REGION Network 57: Step[420] : GapPad Down
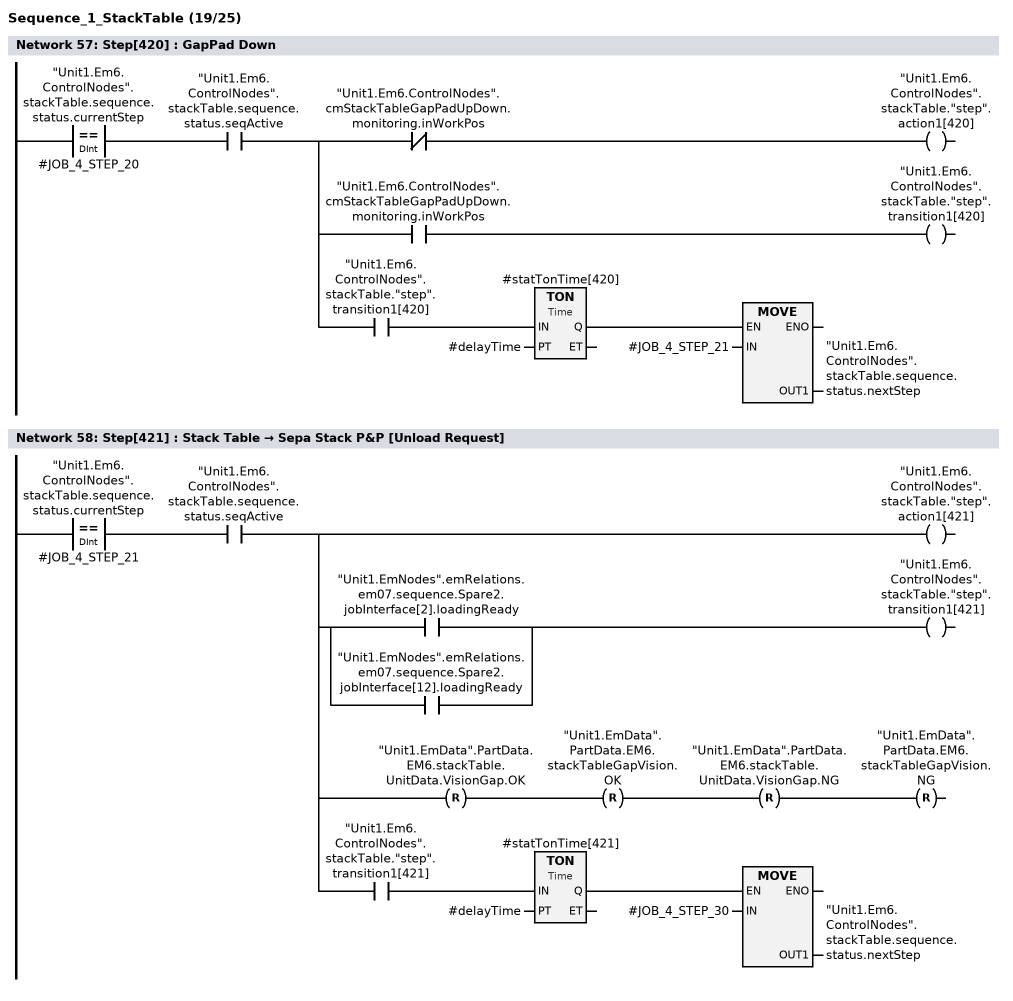
   RUNG wire#powerrail
      { S7_Templates := "SrcType := DInt" } EQ_Contact(in1 := "Unit1.Em6.ControlNodes".stackTable.sequence.status.currentStep, in2 := #JOB_4_STEP_20)
      Contact( "Unit1.Em6.ControlNodes".stackTable.sequence.status.seqActive )
      wire#w1
      I_Contact( "Unit1.Em6.ControlNodes".cmStackTableGapPadUpDown.monitoring.inWorkPos )
      Coil( "Unit1.Em6.ControlNodes".stackTable."step".action1[420] )
   END_RUNG
   RUNG wire#w1
      Contact( "Unit1.Em6.ControlNodes".cmStackTableGapPadUpDown.monitoring.inWorkPos )
      Coil( "Unit1.Em6.ControlNodes".stackTable."step".transition1[420] )
   END_RUNG
   RUNG wire#w1
      Contact( "Unit1.Em6.ControlNodes".stackTable."step".transition1[420] )
      { S7_Templates := "time_type := Time" } #statTonTime[420].TON(pt := #delayTime, et =>)
      Move(in := #JOB_4_STEP_21, out1 => "Unit1.Em6.ControlNodes".stackTable.sequence.status.nextStep)
   END_RUNG
   // the same network as SCL:
   #_w1 := ("Unit1.Em6.ControlNodes".stackTable.sequence.status.currentStep = #JOB_4_STEP_20) AND "Unit1.Em6.ControlNodes".stackTable.sequence.status.seqActive;
   "Unit1.Em6.ControlNodes".stackTable."step".action1[420] := #_w1 AND NOT "Unit1.Em6.ControlNodes".cmStackTableGapPadUpDown.monitoring.inWorkPos;
   "Unit1.Em6.ControlNodes".stackTable."step".transition1[420] := #_w1 AND "Unit1.Em6.ControlNodes".cmStackTableGapPadUpDown.monitoring.inWorkPos;
   #statTonTime[420].TON(IN := #_w1 AND "Unit1.Em6.ControlNodes".stackTable."step".transition1[420],
                         PT := #delayTime);
   IF #statTonTime[420].Q THEN
       "Unit1.Em6.ControlNodes".stackTable.sequence.status.nextStep := #JOB_4_STEP_21;
   END_IF;
END_REGION

REGION Network 58: Step[421] : Stack Table → Sepa Stack P&P [Unload Request]
   RUNG wire#powerrail
      { S7_Templates := "SrcType := DInt" } EQ_Contact(in1 := "Unit1.Em6.ControlNodes".stackTable.sequence.status.currentStep, in2 := #JOB_4_STEP_21)
      Contact( "Unit1.Em6.ControlNodes".stackTable.sequence.status.seqActive )
      wire#w1
      Coil( "Unit1.Em6.ControlNodes".stackTable."step".action1[421] )
   END_RUNG
   RUNG wire#w1
      Contact( "Unit1.EmNodes".emRelations.em07.sequence.Spare2.jobInterface[2].loadingReady )
      wire#w2
      Coil( "Unit1.Em6.ControlNodes".stackTable."step".transition1[421] )
   END_RUNG
   RUNG wire#w1
      Contact( "Unit1.EmNodes".emRelations.em07.sequence.Spare2.jobInterface[12].loadingReady )
   END_RUNG wire#w2
   RUNG wire#w1
      R_Coil( "Unit1.EmData".PartData.EM6.stackTable.UnitData.VisionGap.OK )
      R_Coil( "Unit1.EmData".PartData.EM6.stackTableGapVision.OK )
      R_Coil( "Unit1.EmData".PartData.EM6.stackTable.UnitData.VisionGap.NG )
      R_Coil( "Unit1.EmData".PartData.EM6.stackTableGapVision.NG )
   END_RUNG
   RUNG wire#w1
      Contact( "Unit1.Em6.ControlNodes".stackTable."step".transition1[421] )
      { S7_Templates := "time_type := Time" } #statTonTime[421].TON(pt := #delayTime, et =>)
      Move(in := #JOB_4_STEP_30, out1 => "Unit1.Em6.ControlNodes".stackTable.sequence.status.nextStep)
   END_RUNG
   // the same network as SCL:
   "Unit1.Em6.ControlNodes".stackTable."step".action1[421] := ("Unit1.Em6.ControlNodes".stackTable.sequence.status.currentStep = #JOB_4_STEP_21) AND "Unit1.Em6.ControlNodes".stackTable.sequence.status.seqActive;
   "Unit1.Em6.ControlNodes".stackTable."step".transition1[421] := ("Unit1.Em6.ControlNodes".stackTable.sequence.status.currentStep = #JOB_4_STEP_21) AND "Unit1.Em6.ControlNodes".stackTable.sequence.status.seqActive AND ("Unit1.EmNodes".emRelations.em07.sequence.Spare2.jobInterface[2].loadingReady OR "Unit1.EmNodes".emRelations.em07.sequence.Spare2.jobInterface[12].loadingReady);
   IF ("Unit1.Em6.ControlNodes".stackTable.sequence.status.currentStep = #JOB_4_STEP_21) AND "Unit1.Em6.ControlNodes".stackTable.sequence.status.seqActive THEN
       "Unit1.EmData".PartData.EM6.stackTable.UnitData.VisionGap.OK := FALSE;
       "Unit1.EmData".PartData.EM6.stackTableGapVision.OK := FALSE;
       "Unit1.EmData".PartData.EM6.stackTable.UnitData.VisionGap.NG := FALSE;
       "Unit1.EmData".PartData.EM6.stackTableGapVision.NG := FALSE;
   END_IF;
   #statTonTime[421].TON(IN := ("Unit1.Em6.ControlNodes".stackTable.sequence.status.currentStep = #JOB_4_STEP_21) AND "Unit1.Em6.ControlNodes".stackTable.sequence.status.seqActive AND "Unit1.Em6.ControlNodes".stackTable."step".transition1[421],
                         PT := #delayTime);
   IF #statTonTime[421].Q THEN
       "Unit1.Em6.ControlNodes".stackTable.sequence.status.nextStep := #JOB_4_STEP_30;
   END_IF;
END_REGION

REGION Network 59: Step[430] : A,C.Mendrel Y,Z-Axis Wait Pos
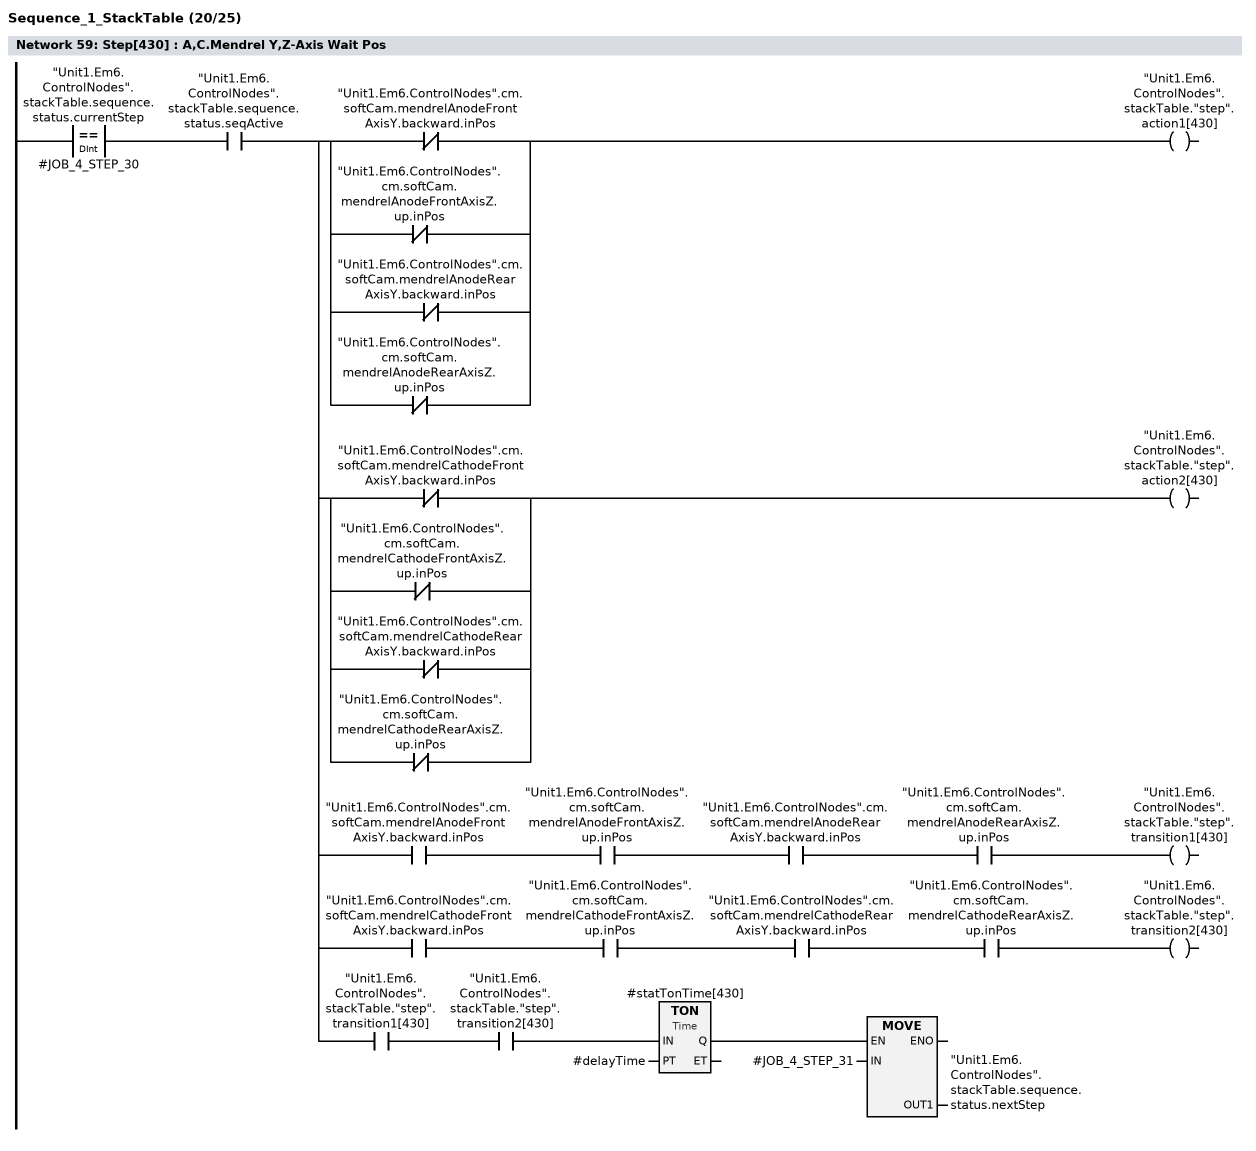
   RUNG wire#powerrail
      { S7_Templates := "SrcType := DInt" } EQ_Contact(in1 := "Unit1.Em6.ControlNodes".stackTable.sequence.status.currentStep, in2 := #JOB_4_STEP_30)
      Contact( "Unit1.Em6.ControlNodes".stackTable.sequence.status.seqActive )
      wire#w1
      I_Contact( "Unit1.Em6.ControlNodes".cm.softCam.mendrelAnodeFrontAxisY.backward.inPos )
      wire#w2
      Coil( "Unit1.Em6.ControlNodes".stackTable."step".action1[430] )
   END_RUNG
   RUNG wire#w1
      I_Contact( "Unit1.Em6.ControlNodes".cm.softCam.mendrelAnodeFrontAxisZ.up.inPos )
   END_RUNG wire#w2
   RUNG wire#w1
      I_Contact( "Unit1.Em6.ControlNodes".cm.softCam.mendrelAnodeRearAxisY.backward.inPos )
   END_RUNG wire#w2
   RUNG wire#w1
      I_Contact( "Unit1.Em6.ControlNodes".cm.softCam.mendrelAnodeRearAxisZ.up.inPos )
   END_RUNG wire#w2
   RUNG wire#w1
      I_Contact( "Unit1.Em6.ControlNodes".cm.softCam.mendrelCathodeFrontAxisY.backward.inPos )
      wire#w3
      Coil( "Unit1.Em6.ControlNodes".stackTable."step".action2[430] )
   END_RUNG
   RUNG wire#w1
      I_Contact( "Unit1.Em6.ControlNodes".cm.softCam.mendrelCathodeFrontAxisZ.up.inPos )
   END_RUNG wire#w3
   RUNG wire#w1
      I_Contact( "Unit1.Em6.ControlNodes".cm.softCam.mendrelCathodeRearAxisY.backward.inPos )
   END_RUNG wire#w3
   RUNG wire#w1
      I_Contact( "Unit1.Em6.ControlNodes".cm.softCam.mendrelCathodeRearAxisZ.up.inPos )
   END_RUNG wire#w3
   RUNG wire#w1
      Contact( "Unit1.Em6.ControlNodes".cm.softCam.mendrelAnodeFrontAxisY.backward.inPos )
      Contact( "Unit1.Em6.ControlNodes".cm.softCam.mendrelAnodeFrontAxisZ.up.inPos )
      Contact( "Unit1.Em6.ControlNodes".cm.softCam.mendrelAnodeRearAxisY.backward.inPos )
      Contact( "Unit1.Em6.ControlNodes".cm.softCam.mendrelAnodeRearAxisZ.up.inPos )
      Coil( "Unit1.Em6.ControlNodes".stackTable."step".transition1[430] )
   END_RUNG
   RUNG wire#w1
      Contact( "Unit1.Em6.ControlNodes".cm.softCam.mendrelCathodeFrontAxisY.backward.inPos )
      Contact( "Unit1.Em6.ControlNodes".cm.softCam.mendrelCathodeFrontAxisZ.up.inPos )
      Contact( "Unit1.Em6.ControlNodes".cm.softCam.mendrelCathodeRearAxisY.backward.inPos )
      Contact( "Unit1.Em6.ControlNodes".cm.softCam.mendrelCathodeRearAxisZ.up.inPos )
      Coil( "Unit1.Em6.ControlNodes".stackTable."step".transition2[430] )
   END_RUNG
   RUNG wire#w1
      Contact( "Unit1.Em6.ControlNodes".stackTable."step".transition1[430] )
      Contact( "Unit1.Em6.ControlNodes".stackTable."step".transition2[430] )
      { S7_Templates := "time_type := Time" } #statTonTime[430].TON(pt := #delayTime, et =>)
      Move(in := #JOB_4_STEP_31, out1 => "Unit1.Em6.ControlNodes".stackTable.sequence.status.nextStep)
   END_RUNG
   // the same network as SCL:
   #_w1 := ("Unit1.Em6.ControlNodes".stackTable.sequence.status.currentStep = #JOB_4_STEP_30) AND "Unit1.Em6.ControlNodes".stackTable.sequence.status.seqActive;
   "Unit1.Em6.ControlNodes".stackTable."step".action1[430] := #_w1 AND (NOT "Unit1.Em6.ControlNodes".cm.softCam.mendrelAnodeFrontAxisY.backward.inPos OR NOT "Unit1.Em6.ControlNodes".cm.softCam.mendrelAnodeFrontAxisZ.up.inPos OR NOT "Unit1.Em6.ControlNodes".cm.softCam.mendrelAnodeRearAxisY.backward.inPos OR NOT "Unit1.Em6.ControlNodes".cm.softCam.mendrelAnodeRearAxisZ.up.inPos);
   "Unit1.Em6.ControlNodes".stackTable."step".action2[430] := #_w1 AND (NOT "Unit1.Em6.ControlNodes".cm.softCam.mendrelCathodeFrontAxisY.backward.inPos OR NOT "Unit1.Em6.ControlNodes".cm.softCam.mendrelCathodeFrontAxisZ.up.inPos OR NOT "Unit1.Em6.ControlNodes".cm.softCam.mendrelCathodeRearAxisY.backward.inPos OR NOT "Unit1.Em6.ControlNodes".cm.softCam.mendrelCathodeRearAxisZ.up.inPos);
   "Unit1.Em6.ControlNodes".stackTable."step".transition1[430] := #_w1 AND "Unit1.Em6.ControlNodes".cm.softCam.mendrelAnodeFrontAxisY.backward.inPos AND "Unit1.Em6.ControlNodes".cm.softCam.mendrelAnodeFrontAxisZ.up.inPos AND "Unit1.Em6.ControlNodes".cm.softCam.mendrelAnodeRearAxisY.backward.inPos AND "Unit1.Em6.ControlNodes".cm.softCam.mendrelAnodeRearAxisZ.up.inPos;
   "Unit1.Em6.ControlNodes".stackTable."step".transition2[430] := #_w1 AND "Unit1.Em6.ControlNodes".cm.softCam.mendrelCathodeFrontAxisY.backward.inPos AND "Unit1.Em6.ControlNodes".cm.softCam.mendrelCathodeFrontAxisZ.up.inPos AND "Unit1.Em6.ControlNodes".cm.softCam.mendrelCathodeRearAxisY.backward.inPos AND "Unit1.Em6.ControlNodes".cm.softCam.mendrelCathodeRearAxisZ.up.inPos;
   #statTonTime[430].TON(IN := #_w1 AND "Unit1.Em6.ControlNodes".stackTable."step".transition1[430] AND "Unit1.Em6.ControlNodes".stackTable."step".transition2[430],
                         PT := #delayTime);
   IF #statTonTime[430].Q THEN
       "Unit1.Em6.ControlNodes".stackTable.sequence.status.nextStep := #JOB_4_STEP_31;
   END_IF;
END_REGION

REGION Network 60: Step[431] : Stack Table → Sepa Stack P&P [Unclamp Done]
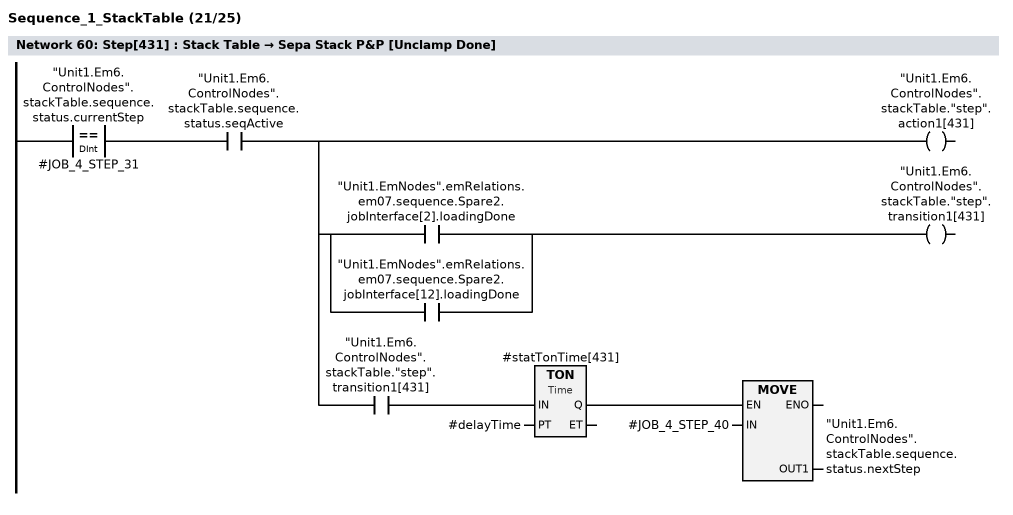
   RUNG wire#powerrail
      { S7_Templates := "SrcType := DInt" } EQ_Contact(in1 := "Unit1.Em6.ControlNodes".stackTable.sequence.status.currentStep, in2 := #JOB_4_STEP_31)
      Contact( "Unit1.Em6.ControlNodes".stackTable.sequence.status.seqActive )
      wire#w1
      Coil( "Unit1.Em6.ControlNodes".stackTable."step".action1[431] )
   END_RUNG
   RUNG wire#w1
      Contact( "Unit1.EmNodes".emRelations.em07.sequence.Spare2.jobInterface[2].loadingDone )
      wire#w2
      Coil( "Unit1.Em6.ControlNodes".stackTable."step".transition1[431] )
   END_RUNG
   RUNG wire#w1
      Contact( "Unit1.EmNodes".emRelations.em07.sequence.Spare2.jobInterface[12].loadingDone )
   END_RUNG wire#w2
   RUNG wire#w1
      Contact( "Unit1.Em6.ControlNodes".stackTable."step".transition1[431] )
      { S7_Templates := "time_type := Time" } #statTonTime[431].TON(pt := #delayTime, et =>)
      Move(in := #JOB_4_STEP_40, out1 => "Unit1.Em6.ControlNodes".stackTable.sequence.status.nextStep)
   END_RUNG
   // the same network as SCL:
   "Unit1.Em6.ControlNodes".stackTable."step".action1[431] := ("Unit1.Em6.ControlNodes".stackTable.sequence.status.currentStep = #JOB_4_STEP_31) AND "Unit1.Em6.ControlNodes".stackTable.sequence.status.seqActive;
   "Unit1.Em6.ControlNodes".stackTable."step".transition1[431] := ("Unit1.Em6.ControlNodes".stackTable.sequence.status.currentStep = #JOB_4_STEP_31) AND "Unit1.Em6.ControlNodes".stackTable.sequence.status.seqActive AND ("Unit1.EmNodes".emRelations.em07.sequence.Spare2.jobInterface[2].loadingDone OR "Unit1.EmNodes".emRelations.em07.sequence.Spare2.jobInterface[12].loadingDone);
   #statTonTime[431].TON(IN := ("Unit1.Em6.ControlNodes".stackTable.sequence.status.currentStep = #JOB_4_STEP_31) AND "Unit1.Em6.ControlNodes".stackTable.sequence.status.seqActive AND "Unit1.Em6.ControlNodes".stackTable."step".transition1[431],
                         PT := #delayTime);
   IF #statTonTime[431].Q THEN
       "Unit1.Em6.ControlNodes".stackTable.sequence.status.nextStep := #JOB_4_STEP_40;
   END_IF;
END_REGION

REGION Network 61: Step[440] : A,C.Mendrel Y,Z-Axis Work Pos
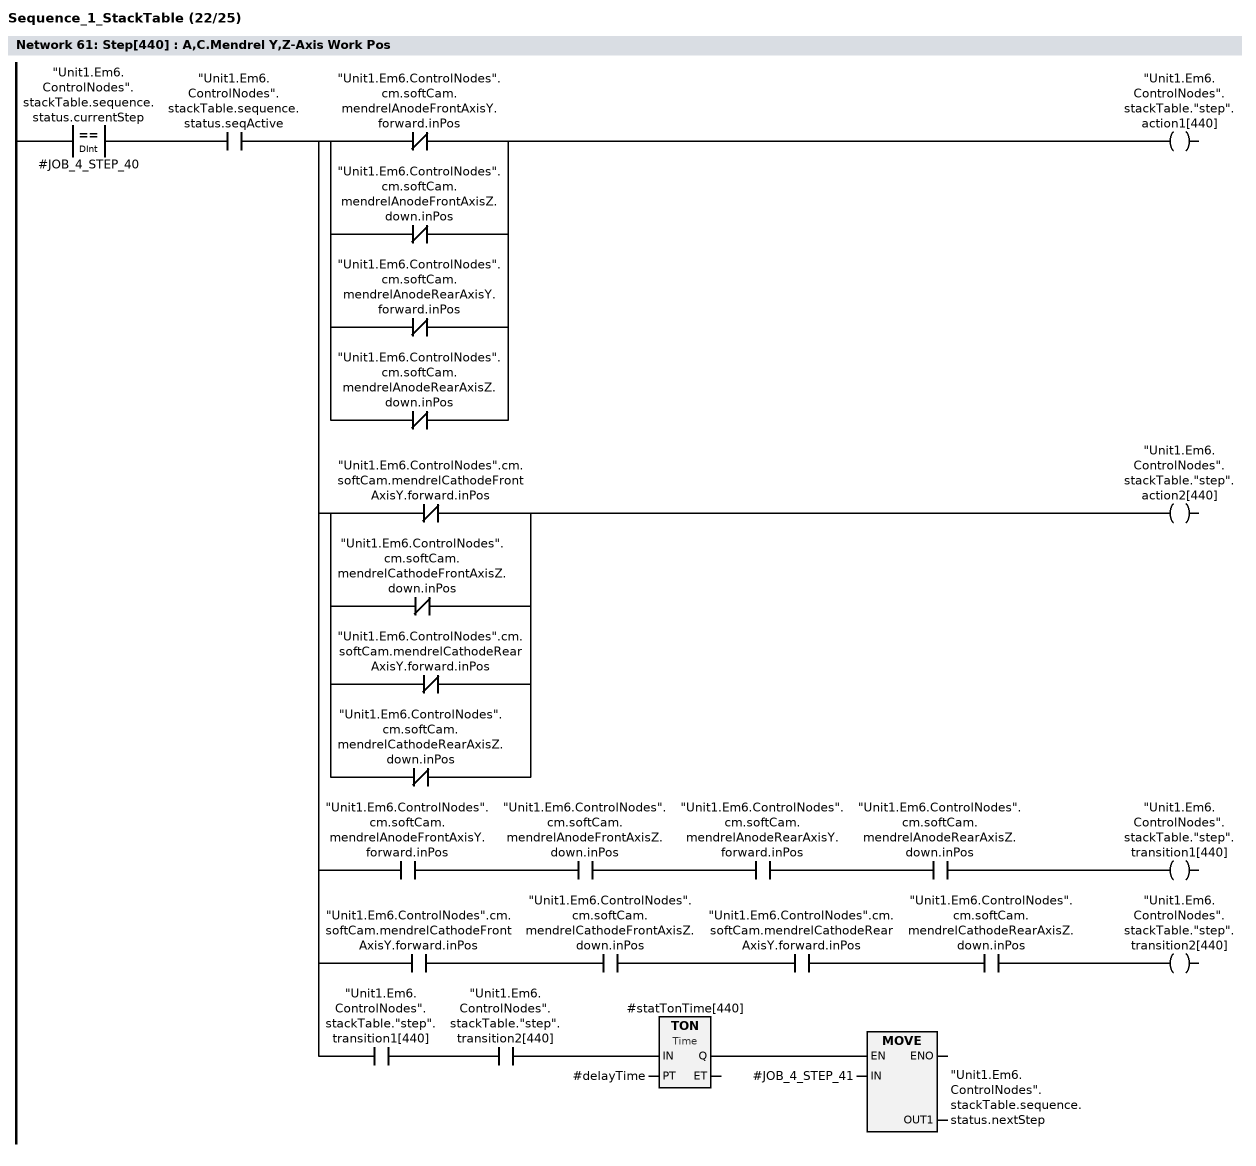
   RUNG wire#powerrail
      { S7_Templates := "SrcType := DInt" } EQ_Contact(in1 := "Unit1.Em6.ControlNodes".stackTable.sequence.status.currentStep, in2 := #JOB_4_STEP_40)
      Contact( "Unit1.Em6.ControlNodes".stackTable.sequence.status.seqActive )
      wire#w1
      I_Contact( "Unit1.Em6.ControlNodes".cm.softCam.mendrelAnodeFrontAxisY.forward.inPos )
      wire#w2
      Coil( "Unit1.Em6.ControlNodes".stackTable."step".action1[440] )
   END_RUNG
   RUNG wire#w1
      I_Contact( "Unit1.Em6.ControlNodes".cm.softCam.mendrelAnodeFrontAxisZ.down.inPos )
   END_RUNG wire#w2
   RUNG wire#w1
      I_Contact( "Unit1.Em6.ControlNodes".cm.softCam.mendrelAnodeRearAxisY.forward.inPos )
   END_RUNG wire#w2
   RUNG wire#w1
      I_Contact( "Unit1.Em6.ControlNodes".cm.softCam.mendrelAnodeRearAxisZ.down.inPos )
   END_RUNG wire#w2
   RUNG wire#w1
      I_Contact( "Unit1.Em6.ControlNodes".cm.softCam.mendrelCathodeFrontAxisY.forward.inPos )
      wire#w3
      Coil( "Unit1.Em6.ControlNodes".stackTable."step".action2[440] )
   END_RUNG
   RUNG wire#w1
      I_Contact( "Unit1.Em6.ControlNodes".cm.softCam.mendrelCathodeFrontAxisZ.down.inPos )
   END_RUNG wire#w3
   RUNG wire#w1
      I_Contact( "Unit1.Em6.ControlNodes".cm.softCam.mendrelCathodeRearAxisY.forward.inPos )
   END_RUNG wire#w3
   RUNG wire#w1
      I_Contact( "Unit1.Em6.ControlNodes".cm.softCam.mendrelCathodeRearAxisZ.down.inPos )
   END_RUNG wire#w3
   RUNG wire#w1
      Contact( "Unit1.Em6.ControlNodes".cm.softCam.mendrelAnodeFrontAxisY.forward.inPos )
      Contact( "Unit1.Em6.ControlNodes".cm.softCam.mendrelAnodeFrontAxisZ.down.inPos )
      Contact( "Unit1.Em6.ControlNodes".cm.softCam.mendrelAnodeRearAxisY.forward.inPos )
      Contact( "Unit1.Em6.ControlNodes".cm.softCam.mendrelAnodeRearAxisZ.down.inPos )
      Coil( "Unit1.Em6.ControlNodes".stackTable."step".transition1[440] )
   END_RUNG
   RUNG wire#w1
      Contact( "Unit1.Em6.ControlNodes".cm.softCam.mendrelCathodeFrontAxisY.forward.inPos )
      Contact( "Unit1.Em6.ControlNodes".cm.softCam.mendrelCathodeFrontAxisZ.down.inPos )
      Contact( "Unit1.Em6.ControlNodes".cm.softCam.mendrelCathodeRearAxisY.forward.inPos )
      Contact( "Unit1.Em6.ControlNodes".cm.softCam.mendrelCathodeRearAxisZ.down.inPos )
      Coil( "Unit1.Em6.ControlNodes".stackTable."step".transition2[440] )
   END_RUNG
   RUNG wire#w1
      Contact( "Unit1.Em6.ControlNodes".stackTable."step".transition1[440] )
      Contact( "Unit1.Em6.ControlNodes".stackTable."step".transition2[440] )
      { S7_Templates := "time_type := Time" } #statTonTime[440].TON(pt := #delayTime, et =>)
      Move(in := #JOB_4_STEP_41, out1 => "Unit1.Em6.ControlNodes".stackTable.sequence.status.nextStep)
   END_RUNG
   // the same network as SCL:
   #_w1 := ("Unit1.Em6.ControlNodes".stackTable.sequence.status.currentStep = #JOB_4_STEP_40) AND "Unit1.Em6.ControlNodes".stackTable.sequence.status.seqActive;
   "Unit1.Em6.ControlNodes".stackTable."step".action1[440] := #_w1 AND (NOT "Unit1.Em6.ControlNodes".cm.softCam.mendrelAnodeFrontAxisY.forward.inPos OR NOT "Unit1.Em6.ControlNodes".cm.softCam.mendrelAnodeFrontAxisZ.down.inPos OR NOT "Unit1.Em6.ControlNodes".cm.softCam.mendrelAnodeRearAxisY.forward.inPos OR NOT "Unit1.Em6.ControlNodes".cm.softCam.mendrelAnodeRearAxisZ.down.inPos);
   "Unit1.Em6.ControlNodes".stackTable."step".action2[440] := #_w1 AND (NOT "Unit1.Em6.ControlNodes".cm.softCam.mendrelCathodeFrontAxisY.forward.inPos OR NOT "Unit1.Em6.ControlNodes".cm.softCam.mendrelCathodeFrontAxisZ.down.inPos OR NOT "Unit1.Em6.ControlNodes".cm.softCam.mendrelCathodeRearAxisY.forward.inPos OR NOT "Unit1.Em6.ControlNodes".cm.softCam.mendrelCathodeRearAxisZ.down.inPos);
   "Unit1.Em6.ControlNodes".stackTable."step".transition1[440] := #_w1 AND "Unit1.Em6.ControlNodes".cm.softCam.mendrelAnodeFrontAxisY.forward.inPos AND "Unit1.Em6.ControlNodes".cm.softCam.mendrelAnodeFrontAxisZ.down.inPos AND "Unit1.Em6.ControlNodes".cm.softCam.mendrelAnodeRearAxisY.forward.inPos AND "Unit1.Em6.ControlNodes".cm.softCam.mendrelAnodeRearAxisZ.down.inPos;
   "Unit1.Em6.ControlNodes".stackTable."step".transition2[440] := #_w1 AND "Unit1.Em6.ControlNodes".cm.softCam.mendrelCathodeFrontAxisY.forward.inPos AND "Unit1.Em6.ControlNodes".cm.softCam.mendrelCathodeFrontAxisZ.down.inPos AND "Unit1.Em6.ControlNodes".cm.softCam.mendrelCathodeRearAxisY.forward.inPos AND "Unit1.Em6.ControlNodes".cm.softCam.mendrelCathodeRearAxisZ.down.inPos;
   #statTonTime[440].TON(IN := #_w1 AND "Unit1.Em6.ControlNodes".stackTable."step".transition1[440] AND "Unit1.Em6.ControlNodes".stackTable."step".transition2[440],
                         PT := #delayTime);
   IF #statTonTime[440].Q THEN
       "Unit1.Em6.ControlNodes".stackTable.sequence.status.nextStep := #JOB_4_STEP_41;
   END_IF;
END_REGION

REGION Network 62: Step[441] : Stack Table → Sepa Stack P&P [Clamp Done]
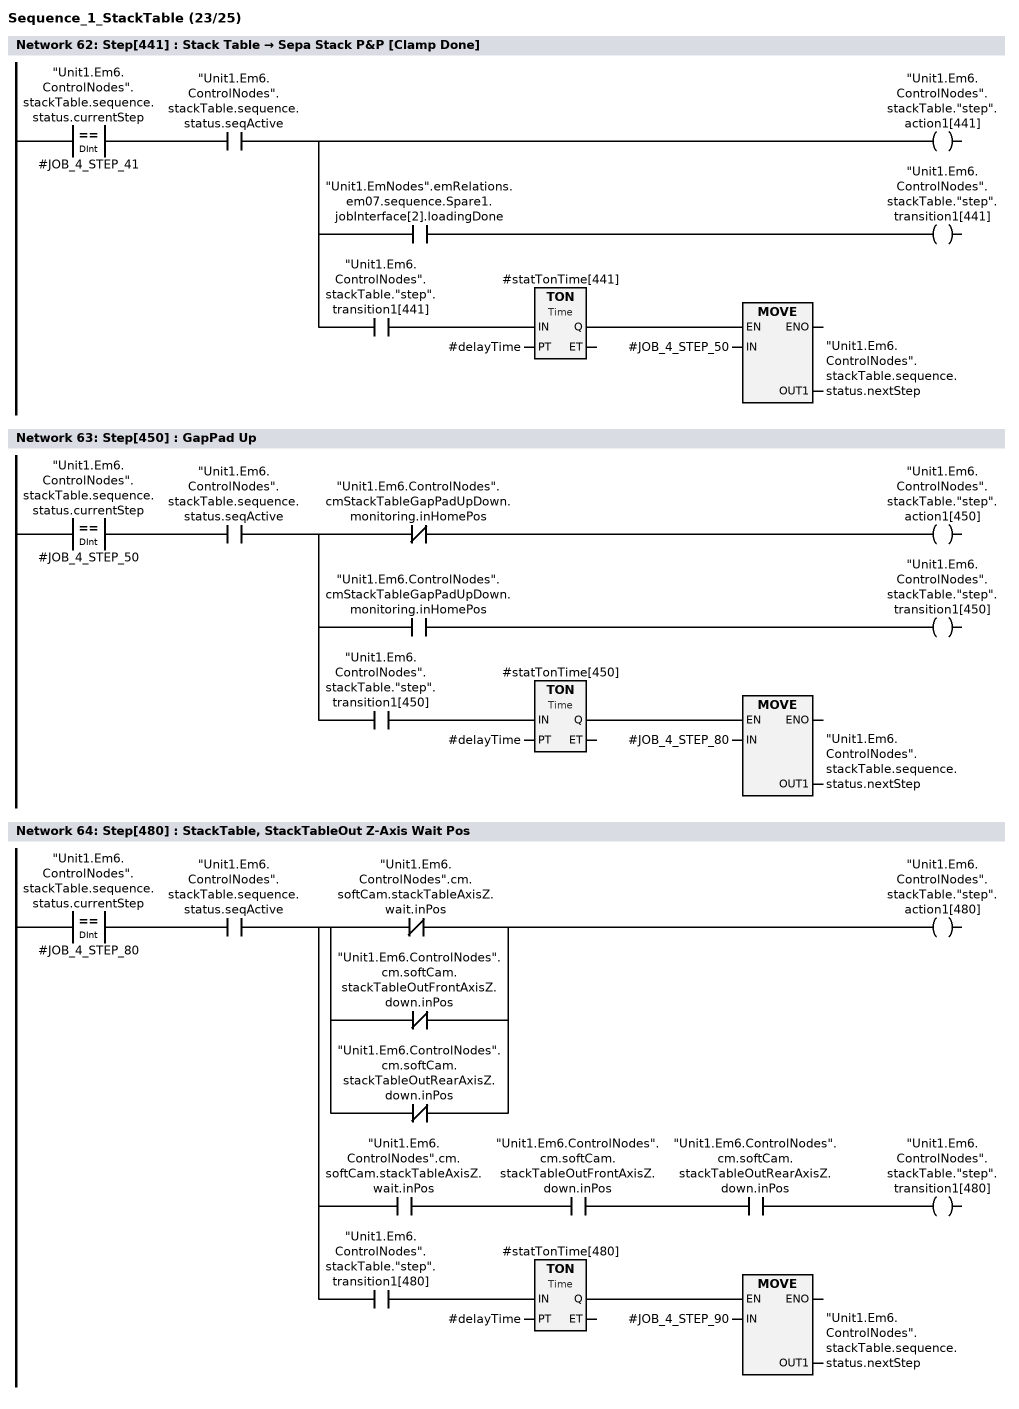
   RUNG wire#powerrail
      { S7_Templates := "SrcType := DInt" } EQ_Contact(in1 := "Unit1.Em6.ControlNodes".stackTable.sequence.status.currentStep, in2 := #JOB_4_STEP_41)
      Contact( "Unit1.Em6.ControlNodes".stackTable.sequence.status.seqActive )
      wire#w1
      Coil( "Unit1.Em6.ControlNodes".stackTable."step".action1[441] )
   END_RUNG
   RUNG wire#w1
      Contact( "Unit1.EmNodes".emRelations.em07.sequence.Spare1.jobInterface[2].loadingDone )
      Coil( "Unit1.Em6.ControlNodes".stackTable."step".transition1[441] )
   END_RUNG
   RUNG wire#w1
      Contact( "Unit1.Em6.ControlNodes".stackTable."step".transition1[441] )
      { S7_Templates := "time_type := Time" } #statTonTime[441].TON(pt := #delayTime, et =>)
      Move(in := #JOB_4_STEP_50, out1 => "Unit1.Em6.ControlNodes".stackTable.sequence.status.nextStep)
   END_RUNG
   // the same network as SCL:
   "Unit1.Em6.ControlNodes".stackTable."step".action1[441] := ("Unit1.Em6.ControlNodes".stackTable.sequence.status.currentStep = #JOB_4_STEP_41) AND "Unit1.Em6.ControlNodes".stackTable.sequence.status.seqActive;
   "Unit1.Em6.ControlNodes".stackTable."step".transition1[441] := ("Unit1.Em6.ControlNodes".stackTable.sequence.status.currentStep = #JOB_4_STEP_41) AND "Unit1.Em6.ControlNodes".stackTable.sequence.status.seqActive AND "Unit1.EmNodes".emRelations.em07.sequence.Spare1.jobInterface[2].loadingDone;
   #statTonTime[441].TON(IN := ("Unit1.Em6.ControlNodes".stackTable.sequence.status.currentStep = #JOB_4_STEP_41) AND "Unit1.Em6.ControlNodes".stackTable.sequence.status.seqActive AND "Unit1.Em6.ControlNodes".stackTable."step".transition1[441],
                         PT := #delayTime);
   IF #statTonTime[441].Q THEN
       "Unit1.Em6.ControlNodes".stackTable.sequence.status.nextStep := #JOB_4_STEP_50;
   END_IF;
END_REGION

REGION Network 63: Step[450] : GapPad Up
   RUNG wire#powerrail
      { S7_Templates := "SrcType := DInt" } EQ_Contact(in1 := "Unit1.Em6.ControlNodes".stackTable.sequence.status.currentStep, in2 := #JOB_4_STEP_50)
      Contact( "Unit1.Em6.ControlNodes".stackTable.sequence.status.seqActive )
      wire#w1
      I_Contact( "Unit1.Em6.ControlNodes".cmStackTableGapPadUpDown.monitoring.inHomePos )
      Coil( "Unit1.Em6.ControlNodes".stackTable."step".action1[450] )
   END_RUNG
   RUNG wire#w1
      Contact( "Unit1.Em6.ControlNodes".cmStackTableGapPadUpDown.monitoring.inHomePos )
      Coil( "Unit1.Em6.ControlNodes".stackTable."step".transition1[450] )
   END_RUNG
   RUNG wire#w1
      Contact( "Unit1.Em6.ControlNodes".stackTable."step".transition1[450] )
      { S7_Templates := "time_type := Time" } #statTonTime[450].TON(pt := #delayTime, et =>)
      Move(in := #JOB_4_STEP_80, out1 => "Unit1.Em6.ControlNodes".stackTable.sequence.status.nextStep)
   END_RUNG
   // the same network as SCL:
   #_w1 := ("Unit1.Em6.ControlNodes".stackTable.sequence.status.currentStep = #JOB_4_STEP_50) AND "Unit1.Em6.ControlNodes".stackTable.sequence.status.seqActive;
   "Unit1.Em6.ControlNodes".stackTable."step".action1[450] := #_w1 AND NOT "Unit1.Em6.ControlNodes".cmStackTableGapPadUpDown.monitoring.inHomePos;
   "Unit1.Em6.ControlNodes".stackTable."step".transition1[450] := #_w1 AND "Unit1.Em6.ControlNodes".cmStackTableGapPadUpDown.monitoring.inHomePos;
   #statTonTime[450].TON(IN := #_w1 AND "Unit1.Em6.ControlNodes".stackTable."step".transition1[450],
                         PT := #delayTime);
   IF #statTonTime[450].Q THEN
       "Unit1.Em6.ControlNodes".stackTable.sequence.status.nextStep := #JOB_4_STEP_80;
   END_IF;
END_REGION

REGION Network 64: Step[480] : StackTable, StackTableOut Z-Axis Wait Pos
   RUNG wire#powerrail
      { S7_Templates := "SrcType := DInt" } EQ_Contact(in1 := "Unit1.Em6.ControlNodes".stackTable.sequence.status.currentStep, in2 := #JOB_4_STEP_80)
      Contact( "Unit1.Em6.ControlNodes".stackTable.sequence.status.seqActive )
      wire#w1
      I_Contact( "Unit1.Em6.ControlNodes".cm.softCam.stackTableAxisZ.wait.inPos )
      wire#w2
      Coil( "Unit1.Em6.ControlNodes".stackTable."step".action1[480] )
   END_RUNG
   RUNG wire#w1
      I_Contact( "Unit1.Em6.ControlNodes".cm.softCam.stackTableOutFrontAxisZ.down.inPos )
   END_RUNG wire#w2
   RUNG wire#w1
      I_Contact( "Unit1.Em6.ControlNodes".cm.softCam.stackTableOutRearAxisZ.down.inPos )
   END_RUNG wire#w2
   RUNG wire#w1
      Contact( "Unit1.Em6.ControlNodes".cm.softCam.stackTableAxisZ.wait.inPos )
      Contact( "Unit1.Em6.ControlNodes".cm.softCam.stackTableOutFrontAxisZ.down.inPos )
      Contact( "Unit1.Em6.ControlNodes".cm.softCam.stackTableOutRearAxisZ.down.inPos )
      Coil( "Unit1.Em6.ControlNodes".stackTable."step".transition1[480] )
   END_RUNG
   RUNG wire#w1
      Contact( "Unit1.Em6.ControlNodes".stackTable."step".transition1[480] )
      { S7_Templates := "time_type := Time" } #statTonTime[480].TON(pt := #delayTime, et =>)
      Move(in := #JOB_4_STEP_90, out1 => "Unit1.Em6.ControlNodes".stackTable.sequence.status.nextStep)
   END_RUNG
   // the same network as SCL:
   #_w1 := ("Unit1.Em6.ControlNodes".stackTable.sequence.status.currentStep = #JOB_4_STEP_80) AND "Unit1.Em6.ControlNodes".stackTable.sequence.status.seqActive;
   "Unit1.Em6.ControlNodes".stackTable."step".action1[480] := #_w1 AND (NOT "Unit1.Em6.ControlNodes".cm.softCam.stackTableAxisZ.wait.inPos OR NOT "Unit1.Em6.ControlNodes".cm.softCam.stackTableOutFrontAxisZ.down.inPos OR NOT "Unit1.Em6.ControlNodes".cm.softCam.stackTableOutRearAxisZ.down.inPos);
   "Unit1.Em6.ControlNodes".stackTable."step".transition1[480] := #_w1 AND "Unit1.Em6.ControlNodes".cm.softCam.stackTableAxisZ.wait.inPos AND "Unit1.Em6.ControlNodes".cm.softCam.stackTableOutFrontAxisZ.down.inPos AND "Unit1.Em6.ControlNodes".cm.softCam.stackTableOutRearAxisZ.down.inPos;
   #statTonTime[480].TON(IN := #_w1 AND "Unit1.Em6.ControlNodes".stackTable."step".transition1[480],
                         PT := #delayTime);
   IF #statTonTime[480].Q THEN
       "Unit1.Em6.ControlNodes".stackTable.sequence.status.nextStep := #JOB_4_STEP_90;
   END_IF;
END_REGION

REGION Network 65: Step[490] : JOB[4] Step End
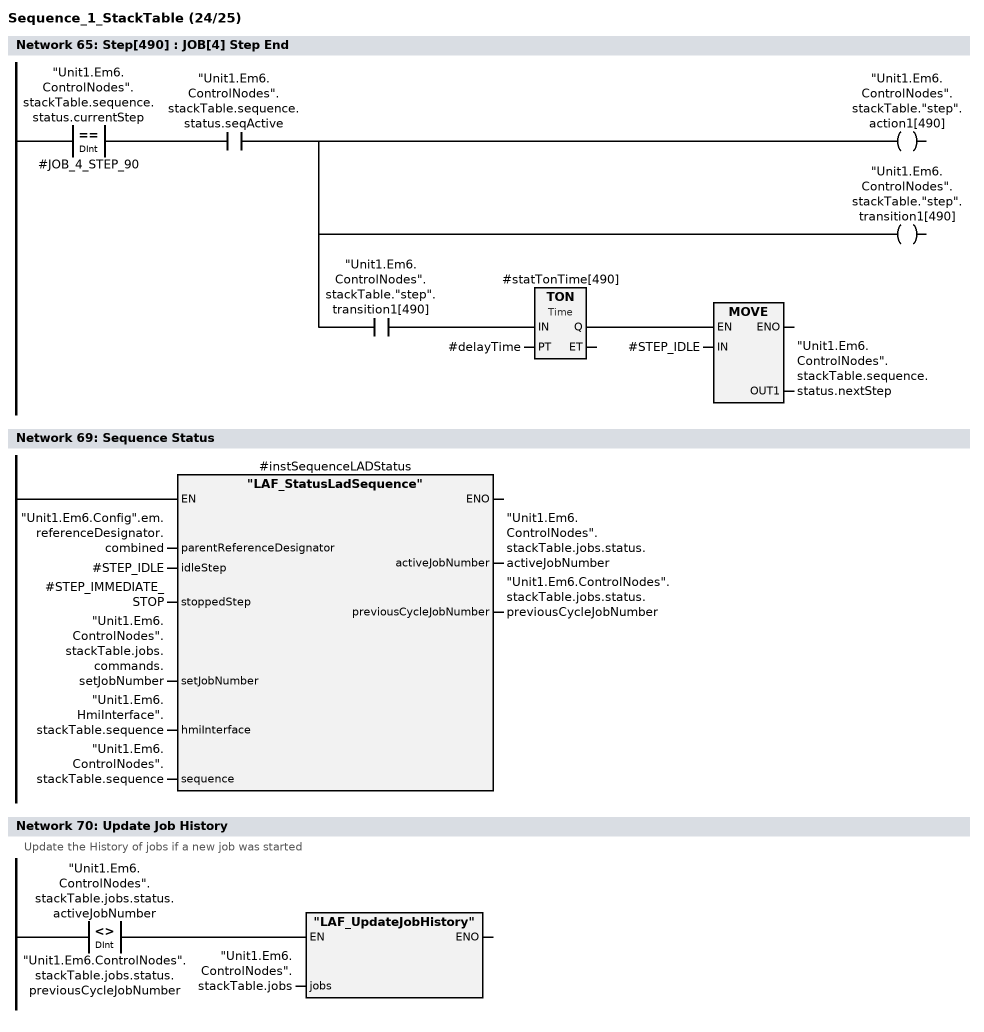
   RUNG wire#powerrail
      { S7_Templates := "SrcType := DInt" } EQ_Contact(in1 := "Unit1.Em6.ControlNodes".stackTable.sequence.status.currentStep, in2 := #JOB_4_STEP_90)
      Contact( "Unit1.Em6.ControlNodes".stackTable.sequence.status.seqActive )
      wire#w1
      Coil( "Unit1.Em6.ControlNodes".stackTable."step".action1[490] )
   END_RUNG
   RUNG wire#w1
      Coil( "Unit1.Em6.ControlNodes".stackTable."step".transition1[490] )
   END_RUNG
   RUNG wire#w1
      Contact( "Unit1.Em6.ControlNodes".stackTable."step".transition1[490] )
      { S7_Templates := "time_type := Time" } #statTonTime[490].TON(pt := #delayTime, et =>)
      Move(in := #STEP_IDLE, out1 => "Unit1.Em6.ControlNodes".stackTable.sequence.status.nextStep)
   END_RUNG
   // the same network as SCL:
   "Unit1.Em6.ControlNodes".stackTable."step".action1[490] := ("Unit1.Em6.ControlNodes".stackTable.sequence.status.currentStep = #JOB_4_STEP_90) AND "Unit1.Em6.ControlNodes".stackTable.sequence.status.seqActive;
   "Unit1.Em6.ControlNodes".stackTable."step".transition1[490] := ("Unit1.Em6.ControlNodes".stackTable.sequence.status.currentStep = #JOB_4_STEP_90) AND "Unit1.Em6.ControlNodes".stackTable.sequence.status.seqActive;
   #statTonTime[490].TON(IN := ("Unit1.Em6.ControlNodes".stackTable.sequence.status.currentStep = #JOB_4_STEP_90) AND "Unit1.Em6.ControlNodes".stackTable.sequence.status.seqActive AND "Unit1.Em6.ControlNodes".stackTable."step".transition1[490],
                         PT := #delayTime);
   IF #statTonTime[490].Q THEN
       "Unit1.Em6.ControlNodes".stackTable.sequence.status.nextStep := #STEP_IDLE;
   END_IF;
END_REGION

REGION Network 66: *************** IMMEDIATE STOP **************************
END_REGION

REGION Network 67: Immediate Stop
END_REGION

REGION Network 68: *************** Status updates **************************
END_REGION

REGION Network 69: Sequence Status
   RUNG wire#powerrail
      #instSequenceLADStatus(parentReferenceDesignator := "Unit1.Em6.Config".em.referenceDesignator.combined, idleStep := #STEP_IDLE, stoppedStep := #STEP_IMMEDIATE_STOP, setJobNumber := "Unit1.Em6.ControlNodes".stackTable.jobs.commands.setJobNumber, hmiInterface := "Unit1.Em6.HmiInterface".stackTable.sequence, sequence := "Unit1.Em6.ControlNodes".stackTable.sequence, activeJobNumber => "Unit1.Em6.ControlNodes".stackTable.jobs.status.activeJobNumber, previousCycleJobNumber => "Unit1.Em6.ControlNodes".stackTable.jobs.status.previousCycleJobNumber)
   END_RUNG
   // the same network as SCL:
   #instSequenceLADStatus(parentReferenceDesignator := "Unit1.Em6.Config".em.referenceDesignator.combined,   // "LAF_StatusLadSequence"
                          idleStep := #STEP_IDLE,
                          stoppedStep := #STEP_IMMEDIATE_STOP,
                          setJobNumber := "Unit1.Em6.ControlNodes".stackTable.jobs.commands.setJobNumber,
                          hmiInterface := "Unit1.Em6.HmiInterface".stackTable.sequence,
                          sequence := "Unit1.Em6.ControlNodes".stackTable.sequence,
                          activeJobNumber => "Unit1.Em6.ControlNodes".stackTable.jobs.status.activeJobNumber,
                          previousCycleJobNumber => "Unit1.Em6.ControlNodes".stackTable.jobs.status.previousCycleJobNumber);
END_REGION

REGION Network 70: Update Job History
   // Update the History of jobs if a new job was started
   RUNG wire#powerrail
      { S7_Templates := "SrcType := DInt" } NE_Contact(in1 := "Unit1.Em6.ControlNodes".stackTable.jobs.status.activeJobNumber, in2 := "Unit1.Em6.ControlNodes".stackTable.jobs.status.previousCycleJobNumber)
      "LAF_UpdateJobHistory"(jobs := "Unit1.Em6.ControlNodes".stackTable.jobs)
   END_RUNG
   // the same network as SCL:
   IF "Unit1.Em6.ControlNodes".stackTable.jobs.status.activeJobNumber <> "Unit1.Em6.ControlNodes".stackTable.jobs.status.previousCycleJobNumber THEN
       "LAF_UpdateJobHistory"(jobs := "Unit1.Em6.ControlNodes".stackTable.jobs);
   END_IF;
END_REGION

REGION Network 71: Output steps as String
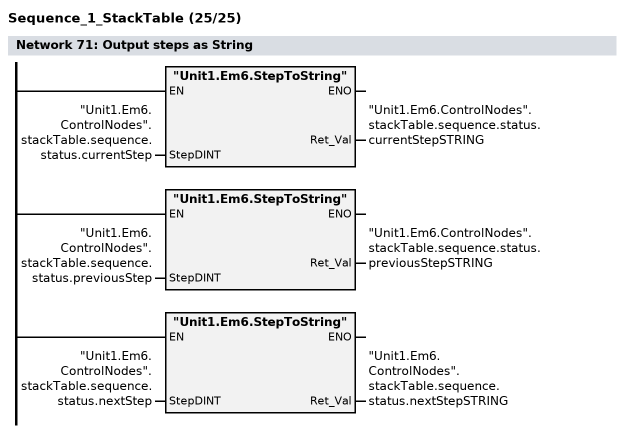
   RUNG wire#powerrail
      "Unit1.Em6.StepToString"(StepDINT := "Unit1.Em6.ControlNodes".stackTable.sequence.status.currentStep, Ret_Val => "Unit1.Em6.ControlNodes".stackTable.sequence.status.currentStepSTRING)
   END_RUNG
   RUNG wire#powerrail
      "Unit1.Em6.StepToString"(StepDINT := "Unit1.Em6.ControlNodes".stackTable.sequence.status.previousStep, Ret_Val => "Unit1.Em6.ControlNodes".stackTable.sequence.status.previousStepSTRING)
   END_RUNG
   RUNG wire#powerrail
      "Unit1.Em6.StepToString"(StepDINT := "Unit1.Em6.ControlNodes".stackTable.sequence.status.nextStep, Ret_Val => "Unit1.Em6.ControlNodes".stackTable.sequence.status.nextStepSTRING)
   END_RUNG
   // the same network as SCL:
   "Unit1.Em6.ControlNodes".stackTable.sequence.status.currentStepSTRING := "Unit1.Em6.StepToString"(StepDINT := "Unit1.Em6.ControlNodes".stackTable.sequence.status.currentStep);
   "Unit1.Em6.ControlNodes".stackTable.sequence.status.previousStepSTRING := "Unit1.Em6.StepToString"(StepDINT := "Unit1.Em6.ControlNodes".stackTable.sequence.status.previousStep);
   "Unit1.Em6.ControlNodes".stackTable.sequence.status.nextStepSTRING := "Unit1.Em6.StepToString"(StepDINT := "Unit1.Em6.ControlNodes".stackTable.sequence.status.nextStep);
END_REGION
END_FUNCTION_BLOCK
